{attribute 'qualified_only'}
{attribute 'strict'}
{attribute 'to_string'}
TYPE MessageArt :
(
	status,
	auftrag,
	daten,
	parameter
);
END_TYPE

(* stored: Version 1.1.0.1, ProductVersion 3.1.4024.12
   DUT MessageArt: Id {68e60b93-01de-4eb8-a57b-67686d1ca216} *)
